// TIA Portal V17 export
// export: Created 2026-04-13T11:12:04.3797839Z, ExportSetting WithDefaults, DisplayName Totally Integrated Automation Portal, DisplayVersion V17 Update 4, DisplayName TIA Portal Openness, DisplayVersion V17 Update 4, DisplayName TIA Portal Version Control Interface, DisplayVersion V17, DisplayName SINAMICS Startdrive Advanced, DisplayVersion V17, DisplayName SINAMICS Startdrive G130, G150, S120, S150, SINAMICS MV, S210, DisplayVersion V17, DisplayName SINAMICS Startdrive G110M, G120, G120C, G120D, G120P, G115D, DisplayVersion V17, DisplayName STEP 7 Professional, DisplayVersion V17 Update 4, DisplayName STEP 7 Safety, DisplayVersion V17, DisplayName WinCC Professional, DisplayVersion V17 Update 4
DATA_BLOCK "SD"   // DB21
{ S7_Optimized_Access := 'TRUE' }
VERSION : 0.1
// stored: AutoNumber true, DBAccessibleFromOPCUA true, DBAccessibleFromWebserver true, IsOnlyStoredInLoadMemory false, IsRetainMemResEnabled false, IsWriteProtectedInAS false, MemoryReserve 100
   VAR
      KS开始喷雾 : Bool;
      JS结束喷雾 : Bool;
      FW复位 : Bool;
      XT系统状态 : String;
      XT系统检测结果 : String;
      XT系统正常 : Bool;
      PW喷雾开始标志 : Bool;
      PW喷雾结束标志 : Bool;
      CL处理物料总量 : Real;
      YX运行时间显示 : String;
   END_VAR
BEGIN
END_DATA_BLOCK
